J6L2xhaXEvNUtwcVArTG9LWC9qNlNsLzVHaG9QK1BvNlAvbGFxci81T3BxZitUcDZqL2txcXQvNU9rcGYrS21KZi9uR052LzdKR1Z2OXZmNFgvamFLZi80bVprditQbzZQL2lwK2YvNHFlb2YrUHBxSC9oWm1XLzRTWmxmK0hsNVQvZ3BLUS80ZVVrdjlnY1hiL2xKTisveVVmRi84S0RRbi9KQ3dtLzA5ZFV2OVhaVnIvV0dkYy8xOXNYdjlkYUYzL1hXZGcvMXhwWWY5ZGJHUC9ZM0pyLzJWMGEvOW9jMnYvYVhWdS8yWnpidjlwYzIvL2JuaDAvMngzY3Y5cmVITC9iMzE2LzNxRmd2OTJnbi8vYzRGLy8zRjlmUDl5ZjMvL2NuMTcvM1IrZWY5Nmc0SC9lNFdHLzNpSGd2OTdpSVQvZjQyRy8zK0toUCtFa0kzL2lKT00vNGVUanYrT21wSC9nWTZILzRPU2ovOTZqWVgvZlpLSy80T1hqditHbG92L2ZvMkgvMzZPaGY5OWtJVC9mWXVDLzN5TWdQOTRpWUgvZVltRC8zMktoLzkrallML2Q0cUEvM3FLaGY5M2hZUC9lWWVCLzNXR2dQOTJpSUgvY29kKy8zYUpnUDkyaTRIL2VZZUMvM3VLaGY5M2k0UC9qazlWLzhORVUvK0Vpb1QvZkk2RS8zeVBpdjk3a0lyL2U1R08vNEtWalA5L2s0Ny9nSktSLzMrV2pmK0RsWTMvZ0phTi8zNlZqditicEpuL0lTUWUveGdmR2Y5UllWVC9aWFJvLzJWMGEvOW5kMi8vYkhsdS8ydDdjdjl1ZkhUL2JYeHkvMjErZGY5d2hIbi9jNFY5LzNlR2dmOTRpWVQvZUltRi8zZUdnLytBalkzL2dwS04vNE9Xa2YrR21aWC9pSnlWLzRhWWxmK0ptNkQva1orYy81R2ZuUCtRblozL2txV2gvNUtqbnYrVnBLWC9tNnlzLzVxcnF2K2hzSy8vbnErdC82U3pzditxdnJ6L29iU3gvNks0c2YrZ3ViUC9wcjIxLzUyM3NQK2l1N2IvcGJxMC81ZXRwZitXcktUL2thV2EvNUNpbFArTW5KSC9oWnFJLzRLUmd2K0FrWVgvZkk2RC8zdU9ndjkzaTMzL2RvZCsvM09FZXY5d2dYVC9jWDEzLzIxOGRQOXRmblQvYlh0eS8ycDVidjlwZDIzL1puVnIvMlJ6YWY5bmRHei9tMHBSLzdRelF2OWphMkwvWDIxai8yQnNZZjlnYTJEL1htdGgvMTFyWC85ZWExNy9XMnRjLzFsb1hmOVhabHovVm1aWi8xcFhXLzhtSnlUL1NsWkkvMUJlVS85b2RHci9hblpxLzJoNWIvOXJlRy8vYlhweS8yeDhkZjlzZ1hqL2M0VjYvMjUvZC85eGduei9kNFNBLzN1SGdQOTZpb2IvZTVDSi80T1lsZitFbFk3L2dwV04vNGVZbFArSmw1TC9qNktkLzR1Wm12K1NwYWIvbjYycy81eXJxZitacmF2L21xbW4vNWVvcHYrYXJhdi9uSzZ4LzY2NXV2K2lzNnovcUx1Mi82aTl0Zityd3JyL3FMNjEvNlM1c3Yra3Viai9wcnk0LzZlOHNmK2d0cXIvbUt1aC81T21vUCtPbzV2L2o2R1cvNCtpbVArR21JNy9ocHFNLzRDUGhQOThpNFAvZVlwKy8zcUtndjk1aDRML2NZRjgvM09FZWY5d2duZi9hM3B6LzJ4OGRQOXJkMjMvYVhodC8ybDdidjlwZG0zL2FIUnIvMloyYS85aWRHai9rMHhSLzY0NFJ2OWphbUgvWW5Cay8yRnVZdjllYldML1gyNWkvMTV0WXY5ZGJHRC9XMnBmLzF0cVhmOWFhbHYvU0VvNy8weEtQLzlkYVYvL1RsdE4vMlJ3YVA5b2VXLy9hSGx2LzJ0M2IvOXZmM1AvYTMxeS8yMkFkdjl0ZzNyL2RJWjIvM3VIZmY5MGhIci9kb2lCLzMyUGl2OTNpb2IvZ1pXTy80R1lqLytGbUpEL2lweVgvNG1jbFArTm9Kci9pNldpLzVDaW8vK1NwS0QvbDdDcS81eTByLytpdHJIL29yV3UvNlcwci8ranI3SC9wTFd2LzZpNHRQK3J1YmYvcWJ1NS82cS91UCt0d0xiL3E3KzAvNlc4dFArcHdMVC9uN3l1LzZLK3NQK2x1SzcvbDZxZy80eWhtUCtKbjVIL2o2S1UvNFNXamYrR21vNy9nSkdFLzRHT2cvOTZpbjcvZDRaLy8zaUtnUDl5aFgzL2NJTjMvM0dDZHY5dGYzTC9hbjF2LzJsNmJ2OXBlVzMvYVhsdS8yZDBhdjltZFd2L2FYaHQvMloxYXY5a2Myai9qRXRSLzdJdVFQOXFabUQvWVc5bC8xOXdaUDlmYkdQL1hteGsvMTFzWWY5Y2FWLy9XMmxlLzFwcFhIZ1x1MDAzZCIsIl90ZWFjaE1ldGhvZCI6eyJfbWV0aG9kVHlwZSI6IkFVVE9NQVRJQyJ9LCJfaXNJZ25vcmVTbmFwc2hvdFBvc2l0aW9uIjpmYWxzZSwiX2lzQXV0b21hdGljTW92ZSI6dHJ1ZSwiX2lzSWdub3JlUm90YXRpb24iOmZhbHNlfQ==]); state(isChildrenLocked=true)
        URCap Boucle de la localisation de caméra (Robotiq_Wrist_Camera, Robotiq Inc.)
          MoveL speed 80 mm/s, acceleration 50 mm/s^2 (useActiveTCP=true) feature=Calib_1
            Waypoint approche: motionParameters(jointSpeed=1.047198 jointAcceleration=1.396263 cartesianSpeed=0.4 cartesianAcceleration=0.508); TCP in base x=-127.51 y=-324.345 z=215.094 mm, rx=-2.2625 ry=-2.1587 rz=0.0418 rad; joints [-89.286, -99.558, -104.123, -65.824, 88.206, -266.16] deg; feature pose in base x=-115.28 y=-376.355 z=-47.016 mm, rx=2.2478 ry=2.1911 rz=0 rad
            Waypoint recup: motionParameters(jointSpeed=1.047198 jointAcceleration=1.396263 cartesianSpeed=0.15 cartesianAcceleration=0.08); TCP in base x=-120.621 y=-324.408 z=153.783 mm, rx=-2.2059 ry=-2.2161 rz=0.0393 rad; joints [-88.063, -107.147, -113.625, -48.801, 88.216, -267.906] deg
            URCap Main (Robotiq_Grippers, Robotiq Inc.) dataModel(position=55.0, force=100.0, speed=52.0, positionInDouble=55.0, forceInDouble=100.0, speedInDouble=52.0, slaveIds=[9], blocking=true)
            Waypoint approche: motionParameters(jointSpeed=1.047198 jointAcceleration=1.396263 cartesianSpeed=0.15 cartesianAcceleration=0.08); TCP in base x=-127.51 y=-324.345 z=215.094 mm, rx=-2.2625 ry=-2.1587 rz=0.0418 rad; joints [-89.286, -99.558, -104.123, -65.824, 88.206, -266.16] deg
            Waypoint post_prise: motionParameters(jointSpeed=1.047198 jointAcceleration=1.396263 cartesianSpeed=0.25 cartesianAcceleration=1.2); TCP in base x=-119.842 y=-320.203 z=232.501 mm, rx=3.123 ry=-0.1407 rz=0.0686 rad; joints [-89.094, -96.9, -102.497, -69.534, 92.351, -173.46] deg; feature pose in base x=-181.238 y=-310.931 z=-23.576 mm, rx=3.1384 ry=-0.0927 rz=0.0029 rad
            var_1 := False
          MoveJ speed 80 deg/s, acceleration 80 deg/s^2 (useActiveTCP=true) feature=Base
            Waypoint pro_placer: TCP in base x=-107.3 y=-316.96 z=388.086 mm, rx=2.2531 ry=2.1366 rz=-0.0153 rad; joints [-86.259, -95.495, -61.717, -110.755, 90.787, -262.768] deg
            Waypoint placer: motionParameters(nextMotionTime=2); TCP in base x=419.643 y=-190.39 z=199.503 mm, rx=0.0407 ry=-3.1155 rz=0.0032 rad; joints [-8.026, -128.275, -65.037, -78.079, 89.395, -279.194] deg
            URCap Main (Robotiq_Grippers, Robotiq Inc.) dataModel(position=0.0, force=0.0, speed=0.0, positionInDouble=0.0, forceInDouble=0.0, speedInDouble=0.0, slaveIds=[9], blocking=true)
            Waypoint post_placer: TCP in base x=168.877 y=-296.689 z=383.757 mm, rx=2.1025 ry=2.2743 rz=-0.0336 rad; joints [-37.687, -96.241, -62.324, -108.977, 88.416, -221.78] deg
            Loop While (checkContinuously=false) expression=digital_in[1]≟ True  and digital_in[2]≟ False
              URCap Dorner Conveyor (DornerConveyor, Advanced Motion - Controls) dataModel(conv=1, oper=2, speed=100)
            Loop Counting (count=100000) loopVariable(name=Boucle_5)
              URCap Dorner Conveyor (DornerConveyor, Advanced Motion - Controls) dataModel(conv=1, oper=2, speed=100)
        URCap Si aucun objet n’est détecté par la caméra (Robotiq_Wrist_Camera, Robotiq Inc.)
          'Optionnel'
  ElseIf digital_in[5]≟ True
    var_1 := True
    Loop While (checkContinuously=false) expression=var_1≟ True
      MoveJ speed 60 deg/s, acceleration 80 deg/s^2 (useActiveTCP=true) feature=Base
        Waypoint Waypoint_1: TCP in base x=-133.008 y=-272.418 z=432.243 mm, rx=-3.0225 ry=-0.0332 rz=-0.2288 rad; joints [-93.401, -100.875, -37.472, -138.494, 98.06, -184.708] deg
      MoveJ speed 60 deg/s, acceleration 80 deg/s^2 (useActiveTCP=true) feature=Base
        Waypoint photo: TCP in base x=-130.985 y=-299.302 z=389.59 mm, rx=-2.5837 ry=-0.1772 rz=-0.0772 rad; joints [-90.403, -121.375, -12.745, -167.534, 90.797, -188.063] deg
